TEXTLIST TransferPanelCmbTxtList
  1 = '1'
  2 = '2'
  3 = '3'
  4 = '4'
   = ''
END_TEXTLIST

(* stored: Version 1.1.0.1, ProductVersion 3.1.4024.4
   TextList TransferPanelCmbTxtList: Id {14bf6c76-d66f-4d89-9e1d-804aaddd5d35} *)
